(* CODESYS project WagoAppDALI.ecp

Project tree, tasks and I/O mapping:
  Steuerung : 750-8202 PFC200 2ETH RS, WAGO, order no. 0750-8202, version 5.14.3.54
    application Application
      libraries: ; WagoAppDALI, 1.3.0.21 (WAGO); VisuDialogs, * (System)
      task PLC_Task (cyclic, interval t#50ms, priority 15) calls PLC_PRG
      task VISU_TASK (cyclic, interval 100 ms, priority 15) calls VisuElems.Visu_Prg
      program PLC_PRG [CFC]
      visualisation Visualization
    Kbus : Kbus, WAGO, version 1.4.0.2
        unmapped channels: K-BUS diagnostics
    MODBUS
      MODBUS : MODBUS, WAGO, order no. n/a, version 1.1.1.15
    Serial
      COM1 : COM1, WAGO, version 0.0.0.19
  text list GlobalTextList
*)

// Steuerung/Application/PLC_PRG
PROGRAM PLC_PRG
VAR
END_VAR

END_PROGRAM

// Steuerung/Application/Visualization
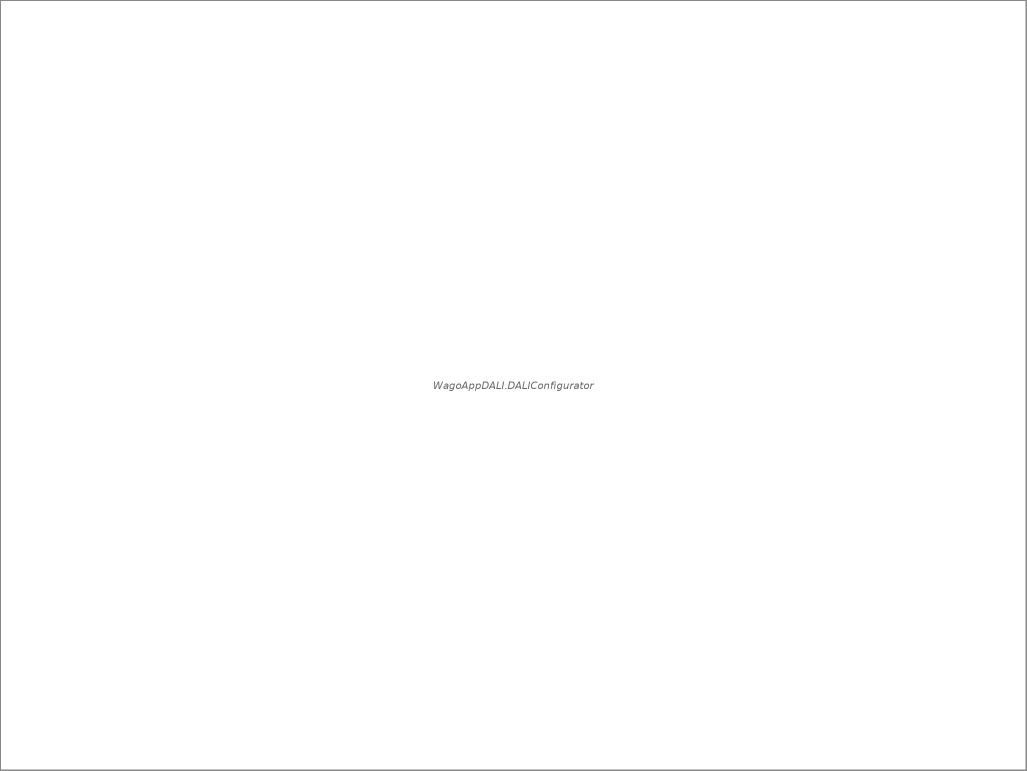
VISUALIZATION Visualization  // 1027x771
    Frame (0,0 1027x771)
        shows WagoAppDALI.DALIConfigurator()
END_VISUALIZATION
